TYPE TupleStruct_2:
    STRUCT
        field0: TupleStruct_1;
        field1: REAL;
    END_STRUCT;
END_TYPE
